Fanuc TP program (LS listing): grp_cls.ls

/PROG  GRP_CLS	  Macro
/ATTR
OWNER		= MNEDITOR;
COMMENT		= "";
PROG_SIZE	= 420;
CREATE		= DATE 19-03-15  TIME 13:58:36;
MODIFIED	= DATE 19-04-15  TIME 15:41:38;
FILE_NAME	= ;
VERSION		= 0;
LINE_COUNT	= 20;
MEMORY_SIZE	= 876;
PROTECT		= READ_WRITE;
TCD:  STACK_SIZE	= 0,
      TASK_PRIORITY	= 50,
      TIME_SLICE	= 0,
      BUSY_LAMP_OFF	= 0,
      ABORT_REQUEST	= 0,
      PAUSE_REQUEST	= 0;
DEFAULT_GROUP	= 1,*,*,*,*;
CONTROL_CODE	= 00000000 00000000;
/MN
   1:  RO[1:Open Gripper]=OFF ;
   2:  RO[2:Close Gripper]=ON ;
   3:   ;
   4:  !Signal to PLC ;
   5:  DO[54]=(RO[2:Close Gripper]) ;
   6:  DO[53]=(RO[1:Open Gripper]) ;
   7:   ;
   8:  WAIT   3.00(sec) ;
   9:   ;
  10:  $WAITTMOUT=200 ;
  11:  WAIT (!RI[1:Gripper Opened]) TIMEOUT,LBL[1] ;
  12:   ;
  13:   ;
  14:  END ;
  15:  LBL[1] ;
  16:  MESSAGE[...] ;
  17:  MESSAGE[GRIPPER] ;
  18:  MESSAGE[NIJE ZATVORIO] ;
  19:  WAIT (!RI[1:Gripper Opened])    ;
  20:  END ;
/POS
/END
